INTERFACE I_CalcXRayTransmission EXTENDS I_Fallible


METHOD Calculate
VAR_INPUT
    MaterialFormula : T_MaxString;
    Thickness : I_QuantityLREAL;
    Transmission : I_QuantityLREALPublic;
END_VAR
END_METHOD

END_INTERFACE

(* stored: Version 1.1.0.1
   Itf I_CalcXRayTransmission: Id {8458f888-4a53-4be0-a69f-01ded61fb385}
   Method Calculate: Id {38d14163-0eee-40ab-9f58-da47106742f3} *)
